TYPE M3TranslationHomingProcedureStatuses :
STRUCT
	///Is the M3GotoProcedure in a busy state?
	busyStatus: BusyStatus;
	///Is the M3GotoProcedure in a healthy state?
	healthStatus: HealthStatus;
END_STRUCT
END_TYPE

(* stored: Version 1.1.0.1, ProductVersion 3.1.4019.2
   DUT M3TranslationHomingProcedureStatuses: Id {b2efa4cf-5090-487d-bc40-ef25f2aebe39} *)
